TYPE Statistics :
STRUCT
	FirstCheck	 :UINT;//首检NG
	His_FirstCheck:UINT;//昨天首检NG
	Hough 		 :UINT;//对齐度NG
	His_Hough    :UINT;//昨天对齐度NG
	JDHough 		 :UINT;//接带对齐度NG
	JDHis_Hough    :UINT;//昨天接带对齐度NG	
	ScanCode	 :UINT;//扫码NG
	ShortTest 	 :UINT;//短路测试NG
	Weight 		 :UINT;//称重NG
	Thickness 	 :UINT;//测厚NG
	MES          :UINT;//MES的NG
	Hough_DT  :ARRAY[1..3] OF UINT;//每个叠台对齐度NG数量
	His_HoughAn  :ARRAY[1..3] OF UINT;//每个叠台对齐度NG正极片数
	His_HoughCa  :ARRAY[1..3] OF UINT;//每个叠台对齐度NG负极片数
END_STRUCT
END_TYPE

(* stored: Version 1.1.0.1, ProductVersion 3.1.4024.12
   DUT Statistics: Id {00e24f56-50c8-43c0-a07d-c6ed5d08d2d2} *)
